{attribute 'pack_mode' := '1'}
TYPE ST_Complex_8 :
STRUCT
	stComplex		: ST_Complex_1;
	strString5		: STRING[5]; (*String, max 5 chars*)
	eEnum	 		: E_Enum_1;
	strString3	 	: STRING[3]; (*String, max 3 chars*)
	arrComplex 		: ARRAY[0..1] OF ST_Complex_1;
	arrDint		 	: ARRAY[0..100] OF DINT;	
END_STRUCT
END_TYPE

(* stored: Version 1.1.0.1
   DUT ST_Complex_8: Id {bc101f5a-7b54-46ec-a90c-0554f2f44d7b} *)
